// TwinCAT 3 PLC project TcSpeech_FbPlay
// ProgramVersion: 3.1.4026.9
// libraries:
//   Tc2_Standard, * (Beckhoff Automation GmbH)
//   Tc2_System, * (Beckhoff Automation GmbH)
//   Tc3_Speech, * (Beckhoff Automation GmbH)
// project tree:
//   / PlcTask.TcTTO
//   POUs/ MAIN.TcPOU, MainPlay.TcPOU
// real-time tasks:
//   TASK PlcTask: cycle T#10ms, priority 20, ADS port 350

CONFIGURATION TcSpeech_FbPlay
    RESOURCE PLC ON TwinCAT3
        TASK PlcTask(INTERVAL := T#10ms, PRIORITY := 20);
        PROGRAM MAIN WITH PlcTask : MAIN;
    END_RESOURCE
END_CONFIGURATION

// ---- POUs/MAIN.TcPOU
PROGRAM MAIN
VAR
END_VAR

MainPlay();

END_PROGRAM

// ---- POUs/MainPlay.TcPOU
PROGRAM MainPlay
VAR
	// fbPlay Variables
	bPlay	: BOOL;
	nConfigId	: UINT := 200;
	sFilePath : STRING(4095) := 'C:\16bit_16khz_mono_SampleSound.wav';
	fbPlay : FB_Play;
	
END_VAR

// Set bPlay to true, to start playback of file
IF bPlay THEN
	fbPlay(bPlay := TRUE, sPath := sFilePath, nConfigurationId := nConfigId);
	
	IF NOT fbPlay.bBusy THEN
		fbPlay(bPlay := FALSE, sPath := sFilePath, nConfigurationId := nConfigId);
		bPlay := FALSE;
	END_IF
END_IF

END_PROGRAM
